(* PLC project Unnamed, Unknown Unnamed 1 *)
(* stored: creationDateTime 2026-03-25T22:12:10, modificationDateTime 2026-03-25T22:12:10 *)

PROGRAM main
  VAR
    WS2812_Out AT %QX0.0 : BOOL;
  END_VAR
  VAR
    BlinkTimer : TON;
    LED_State : BOOL := FALSE;
  END_VAR

            (* 1. 1초 타이머 설정: BlinkTimer.Q가 False일 때 작동 시작, 1초 후 True 반환 *)
BlinkTimer(IN := NOT BlinkTimer.Q, PT := T#1s);

(* 2. 타이머가 완료(1초 경과)될 때마다 실행 *)
IF BlinkTimer.Q THEN
    (* 내부 상태 값을 반전 (False -> True -> False) *)
    LED_State := NOT LED_State;
END_IF;

(* 3. 실제 아두이노 13번 핀(%QX0.6)으로 신호 전송 *)
WS2812_Out := LED_State;
          
END_PROGRAM

CONFIGURATION Config0
  RESOURCE Res0 ON PLC
    TASK task0(INTERVAL := T#20ms, PRIORITY := 1);
    PROGRAM instance0 WITH task0 : main;
  END_RESOURCE
END_CONFIGURATION
